INTERFACE I_Drive_Type_1_Controller

END_INTERFACE

(* stored: Version 1.1.0.1, ProductVersion 3.1.4024.15
   Itf I_Drive_Type_1_Controller: Id {fea85449-4abf-4c82-91ef-68f80e7d266e} *)
